(* Logix 5000 project; controller AplicacionAFEbancoDePruebas vendor 1 type 14 code 149 rev 33.12; software revision 33.01 *)

TASK MainTask (continuous, watchdog 500 ms) : MainProgram

MODULES
   Local : vendor 1 type 14 code 149 (Compact 0, rev 33.12)
      Discrete_IO : Embedded (Compact 1, rev 3.1, Output RPI 20 ms)
      PLC : 1769-L32E Ethernet Port (Ethernet 192.168.2.131, rev 20.1)
         PLC_Controller : vendor 1 type 14 code 77 (CompactLogixL32EController 0, rev 20.1, $1e2c146d$ RPI 20 ms, $44551a5c$ RPI 20 ms, $f7b069ef$ RPI 20 ms)
      VSD_AFE : vendor 1 type 143 code 8336 (Ethernet 192.168.2.50, rev 6.5, Output RPI 20 ms)
           VSD_AFE:O.LogicCommand_Stop   // Comando de Parada
           VSD_AFE:O.LogicCommand_Start   // Comando de Arranque
          : vendor 1 type 143 code 1441 (RhinoBP 10, rev 1.1)
          : vendor 1 type 143 code 416 (RhinoBP 5, rev 1.8)
          : vendor 1 type 143 code 675 (RhinoBP 13, rev 1.1)
          : vendor 1 type 143 code 416 (RhinoBP 4, rev 1.8)
          : vendor 1 type 143 code 4770 (RhinoBP 12, rev 1.1)
          : vendor 1 type 143 code 2724 (RhinoBP 14, rev 1.1)
          : vendor 1 type 143 code 767 (RhinoBP 1, rev 2.7)
END_MODULES

TYPE Dinagrama :   // Estructura para el dinagrama
STRUCT
   vPotencia : REAL[500];   // captura del vector de potencia
   vCarga : REAL[500];   // captura del vector de carga
   vPosicion : REAL[500];   // captura del vector posicion
   vProximetro : DINT[500];   // captura del vector del proximetro
   NumeroMuestras : INT;
   enabled : BOOL;
   captura : BOOL;   // Flag que indica la captura del sistema
   resetVector : BOOL;   // Flag para darle Reset al vector de posición y carga
   vEmptyREAL : REAL[500];
   vEmptyINT : DINT[500];
   tMuestreo : REAL;   // Tiempo de Muestreo de captura
END_STRUCT
END_TYPE

TYPE LSW :   // Drive - Logic Status Word
STRUCT
   Faulted : BOOL;
   Warning : BOOL;
   RunForward : BOOL;
   RunReverse : BOOL;
   Ready : BOOL;
   RemoteRef : BOOL;
   RemoteCrtl : BOOL;
   AtSpeed : BOOL;
END_STRUCT
END_TYPE

TYPE SWC :
STRUCT
   Dinagrama : Dinagrama;
   VSD : VSD;
   entradasDigitales : INT;   // Entradas Digitales
   salidasDigitales : INT;   // Salidas Digitales
   entradasAnalogas : REAL[4];   // Entradas Analogas del PLC
   salidasAnalogas : REAL[4];
END_STRUCT
END_TYPE

TYPE VSD :   // VSD
STRUCT
   VSD_O : AB:PowerFlex755T_E_31635488:O:0;
   VSD_I : AB:PowerFlex755T_E_2B0A69C5:I:0;
END_STRUCT
END_TYPE

VAR_GLOBAL   (* controller tags *)
   SRP_Displacement_Actual : REAL := 47.925312;   // Variable de Simulacion PLC DC de Desplazamiento
   SRP_Load_Actual : REAL := 10.571887;   // Variable de simulacion PLC DC de Carga
   SRP_SimActualStroke : DINT;   // Variable Simulación de PLC Variador DC
   SWC : SWC := (Dinagrama.vCarga[0] := 9.6614, Dinagrama.vCarga[1] := 9.7812, Dinagrama.vCarga[2] := 9.711983, Dinagrama.vCarga[3] := 9.725293, Dinagrama.vCarga[4] := 9.842433, Dinagrama.vCarga[5] := 9.749254, Dinagrama.vCarga[6] := 9.69601, Dinagrama.vCarga[7] := 9.7306185, Dinagrama.vCarga[8] := 9.586858, Dinagrama.vCarga[9] := 9.751916, Dinagrama.vCarga[10] := 10.223133, Dinagrama.vCarga[11] := 10.473384, Dinagrama.vCarga[12] := 10.545264, Dinagrama.vCarga[13] := 10.752919, Dinagrama.vCarga[14] := 10.928628, Dinagrama.vCarga[15] := 11.220809, Dinagrama.vCarga[16] := 11.419147, Dinagrama.vCarga[17] := 11.515653, Dinagrama.vCarga[18] := 11.572558, Dinagrama.vCarga[19] := 11.751262, Dinagrama.vCarga[20] := 11.839782, Dinagrama.vCarga[21] := 11.974224, Dinagrama.vCarga[22] := 11.854091, Dinagrama.vCarga[23] := 11.607167, Dinagrama.vCarga[24] := 11.27239, Dinagrama.vCarga[25] := 11.069394, Dinagrama.vCarga[26] := 10.880708, Dinagrama.vCarga[27] := 10.662403, Dinagrama.vCarga[28] := 10.492021, Dinagrama.vCarga[29] := 10.321636, Dinagrama.vCarga[30] := 10.193849, Dinagrama.vCarga[31] := 10.018141, Dinagrama.vCarga[32] := 9.842432, Dinagrama.vCarga[33] := 9.682698, Dinagrama.vCarga[34] := 9.586857, Dinagrama.vCarga[35] := 9.706658, Dinagrama.vCarga[36] := 9.938273, Dinagrama.vCarga[37] := 10.082034, Dinagrama.vCarga[38] := 10.241769, Dinagrama.vCarga[39] := 10.321636, Dinagrama.vCarga[40] := 10.409491, Dinagrama.vCarga[41] := 10.409491, Dinagrama.vCarga[42] := 10.457411, Dinagrama.vCarga[43] := 10.534616, Dinagrama.vCarga[44] := 10.481371, Dinagrama.vCarga[45] := 10.555914, Dinagrama.vCarga[46] := 10.705, Dinagrama.vCarga[47] := 10.603834, Dinagrama.vCarga[48] := 10.316312, Dinagrama.vCarga[49] := 10.060737, Dinagrama.vCarga[50] := 9.9223, Dinagrama.vCarga[51] := 9.850419, Dinagrama.vCarga[52] := 9.608155, Dinagrama.vCarga[53] := 9.405825, Dinagrama.vCarga[54] := 9.389851, Dinagrama.vCarga[55] := 9.230116, Dinagrama.vCarga[56] := 9.131613, Dinagrama.vCarga[57] := 9.049084, Dinagrama.vCarga[58] := 9.08103, Dinagrama.vCarga[59] := 8.9266205,
        Dinagrama.vCarga[60] := 8.873376, Dinagrama.vCarga[61] := 9.155573, Dinagrama.vCarga[62] := 9.427122, Dinagrama.vCarga[63] := 9.549585, Dinagrama.vCarga[64] := 9.682697, Dinagrama.vCarga[65] := 9.906326, Dinagrama.vCarga[66] := 10.012816, Dinagrama.vCarga[67] := 9.980869, Dinagrama.vCarga[68] := 9.996842, Dinagrama.vCarga[69] := 9.980869, Dinagrama.vCarga[70] := 10.018141, Dinagrama.vCarga[71] := 10.042101, Dinagrama.vCarga[72] := 10.098008, Dinagrama.vCarga[73] := 10.193849, Dinagrama.vCarga[74] := 9.938273, Dinagrama.vCarga[75] := 9.618804, Dinagrama.vCarga[76] := 9.546924, Dinagrama.vCarga[77] := 9.55491, Dinagrama.vCarga[78] := 9.331282, Dinagrama.vCarga[79] := 9.171547, Dinagrama.vCarga[80] := 9.347255, Dinagrama.vCarga[81] := 9.315308, Dinagrama.vCarga[82] := 9.123626, Dinagrama.vCarga[83] := 9.18752, Dinagrama.vCarga[84] := 9.331282, Dinagrama.vCarga[85] := 9.182196, Dinagrama.vCarga[86] := 9.2168045, Dinagrama.vCarga[87] := 9.565559, Dinagrama.vCarga[88] := 9.762566, Dinagrama.vCarga[89] := 9.714645, Dinagrama.vCarga[90] := 9.703996, Dinagrama.vCarga[91] := 9.842432, Dinagrama.vCarga[92] := 9.834445, Dinagrama.vCarga[93] := 9.634777, Dinagrama.vCarga[94] := 9.634777, Dinagrama.vCarga[95] := 9.656075, Dinagrama.vCarga[96] := 9.496341, Dinagrama.vCarga[97] := 9.272713, Dinagrama.vCarga[98] := 9.128951, Dinagrama.vCarga[99] := 8.910647, Dinagrama.vCarga[100] := 8.434105, Dinagrama.vCarga[101] := 8.02412, Dinagrama.vCarga[102] := 7.904319, Dinagrama.vCarga[103] := 7.78718, Dinagrama.vCarga[104] := 7.5129685, Dinagrama.vCarga[105] := 7.302651, Dinagrama.vCarga[106] := 7.281353, Dinagrama.vCarga[107] := 7.238757, Dinagrama.vCarga[108] := 6.8181233, Dinagrama.vCarga[109] := 6.6264415, Dinagrama.vCarga[110] := 6.6796865, Dinagrama.vCarga[111] := 6.903315, Dinagrama.vCarga[112] := 7.1056457, Dinagrama.vCarga[113] := 7.3771944, Dinagrama.vCarga[114] := 7.773869, Dinagrama.vCarga[115] := 7.909643, Dinagrama.vCarga[116] := 7.909643, Dinagrama.vCarga[117] := 8.077365, Dinagrama.vCarga[118] := 8.300993, Dinagrama.vCarga[119] := 8.340926,
        Dinagrama.vCarga[120] := 8.460728, Dinagrama.vCarga[121] := 8.70033, Dinagrama.vCarga[122] := 8.79617, Dinagrama.vCarga[123] := 8.788184, Dinagrama.vCarga[124] := 8.77221, Dinagrama.vCarga[125] := 8.588515, Dinagrama.vCarga[126] := 8.38086, Dinagrama.vCarga[127] := 8.340927, Dinagrama.vCarga[128] := 8.468715, Dinagrama.vCarga[129] := 8.399496, Dinagrama.vCarga[130] := 8.476701, Dinagrama.vCarga[131] := 8.532608, Dinagrama.vCarga[132] := 8.497999, Dinagrama.vCarga[133] := 8.503324, Dinagrama.vCarga[134] := 8.591178, Dinagrama.vCarga[135] := 8.56988, Dinagrama.vCarga[136] := 8.631111, Dinagrama.vCarga[137] := 8.84409, Dinagrama.vCarga[138] := 9.081031, Dinagrama.vCarga[139] := 9.278037, Dinagrama.vCarga[140] := 9.325957, Dinagrama.vCarga[141] := 9.363229, Dinagrama.vCarga[142] := 9.618804, Dinagrama.vCarga[143] := 9.682698, Dinagrama.vCarga[144] := 9.682698, Dinagrama.vCarga[145] := 9.938273, Dinagrama.vCarga[146] := 9.938273, Dinagrama.vCarga[147] := 9.938273, Dinagrama.vCarga[148] := 9.938273, Dinagrama.vCarga[149] := 9.938273, Dinagrama.vCarga[150] := 9.938273, Dinagrama.vCarga[151] := 9.938273, Dinagrama.vCarga[152] := 9.938273, Dinagrama.vCarga[153] := 9.938273, Dinagrama.vCarga[154] := 9.938273, Dinagrama.vCarga[155] := 9.938273, Dinagrama.vCarga[156] := 9.938273, Dinagrama.vCarga[157] := 9.938273, Dinagrama.vCarga[158] := 9.938273, Dinagrama.vCarga[159] := 9.938273, Dinagrama.vCarga[160] := 9.938273, Dinagrama.vCarga[161] := 9.938273, Dinagrama.vCarga[162] := 9.938273, Dinagrama.vCarga[163] := 9.938273, Dinagrama.vCarga[164] := 9.938273, Dinagrama.vCarga[165] := 9.938273, Dinagrama.vCarga[166] := 9.938273, Dinagrama.vCarga[167] := 9.938273, Dinagrama.vCarga[168] := 9.938273, Dinagrama.vCarga[169] := 9.938273, Dinagrama.vCarga[170] := 9.938273, Dinagrama.vCarga[171] := 9.938273, Dinagrama.vCarga[172] := 9.938273, Dinagrama.vCarga[173] := 9.938273, Dinagrama.vCarga[174] := 9.938273, Dinagrama.vCarga[175] := 9.938273, Dinagrama.vCarga[176] := 9.938273, Dinagrama.vCarga[177] := 9.938273, Dinagrama.vCarga[178] := 9.938273, Dinagrama.vCarga[179] := 9.938273,
        Dinagrama.vCarga[180] := 9.938273, Dinagrama.vCarga[181] := 9.938273, Dinagrama.vCarga[182] := 9.938273, Dinagrama.vCarga[183] := 9.938273, Dinagrama.vCarga[184] := 9.938273, Dinagrama.vCarga[185] := 9.938273, Dinagrama.vCarga[186] := 9.938273, Dinagrama.vCarga[187] := 9.938273, Dinagrama.vCarga[188] := 9.938273, Dinagrama.vCarga[189] := 9.938273, Dinagrama.vCarga[190] := 9.938273, Dinagrama.vCarga[191] := 9.938273, Dinagrama.vCarga[192] := 9.938273, Dinagrama.vCarga[193] := 9.938273, Dinagrama.vCarga[194] := 9.938273, Dinagrama.vCarga[195] := 9.938273, Dinagrama.vCarga[196] := 9.938273, Dinagrama.vCarga[197] := 9.938273, Dinagrama.vCarga[198] := 9.938273, Dinagrama.vCarga[199] := 9.938273, Dinagrama.vCarga[200] := 9.938273, Dinagrama.vCarga[201] := 9.938273, Dinagrama.vCarga[202] := 9.938273, Dinagrama.vCarga[203] := 9.938273, Dinagrama.vCarga[204] := 9.938273, Dinagrama.vCarga[205] := 9.938273, Dinagrama.vCarga[206] := 9.938273, Dinagrama.vCarga[207] := 9.938273, Dinagrama.vCarga[208] := 9.938273, Dinagrama.vCarga[209] := 9.938273, Dinagrama.vCarga[210] := 9.938273, Dinagrama.vCarga[211] := 9.938273, Dinagrama.vCarga[212] := 9.938273, Dinagrama.vCarga[213] := 9.938273, Dinagrama.vCarga[214] := 9.938273, Dinagrama.vCarga[215] := 9.938273, Dinagrama.vCarga[216] := 9.938273, Dinagrama.vCarga[217] := 9.938273, Dinagrama.vCarga[218] := 9.938273, Dinagrama.vCarga[219] := 9.938273, Dinagrama.vCarga[220] := 9.938273, Dinagrama.vCarga[221] := 9.938273, Dinagrama.vCarga[222] := 9.938273, Dinagrama.vCarga[223] := 9.938273, Dinagrama.vCarga[224] := 9.938273, Dinagrama.vCarga[225] := 9.938273, Dinagrama.vCarga[226] := 9.938273, Dinagrama.vCarga[227] := 9.938273, Dinagrama.vCarga[228] := 9.938273, Dinagrama.vCarga[229] := 9.938273, Dinagrama.vCarga[230] := 9.938273, Dinagrama.vCarga[231] := 10.060737, Dinagrama.vCarga[232] := 9.9223, Dinagrama.vCarga[233] := 9.7306185, Dinagrama.vCarga[234] := 9.480367, Dinagrama.vCarga[235] := 9.405825, Dinagrama.vCarga[236] := 9.389851, Dinagrama.vCarga[237] := 9.230116, Dinagrama.vCarga[238] := 9.059732, Dinagrama.vCarga[239] := 9.10499,
        Dinagrama.vCarga[240] := 9.017137, Dinagrama.vCarga[241] := 8.822793, Dinagrama.vCarga[242] := 9.0011635, Dinagrama.vCarga[243] := 9.323295, Dinagrama.vCarga[244] := 9.499002, Dinagrama.vCarga[245] := 9.549585, Dinagrama.vCarga[246] := 9.682697, Dinagrama.vCarga[247] := 10.002167, Dinagrama.vCarga[248] := 10.012816, Dinagrama.vCarga[249] := 9.980869, Dinagrama.vCarga[250] := 9.986194, Dinagrama.vCarga[251] := 9.980869, Dinagrama.vCarga[252] := 10.018141, Dinagrama.vCarga[253] := 10.042101, Dinagrama.vCarga[254] := 10.145928, Dinagrama.vCarga[255] := 10.066061, Dinagrama.vCarga[256] := 9.778539, Dinagrama.vCarga[257] := 9.578871, Dinagrama.vCarga[258] := 9.546924, Dinagrama.vCarga[259] := 9.443096, Dinagrama.vCarga[260] := 9.331282, Dinagrama.vCarga[261] := 9.259401, Dinagrama.vCarga[262] := 9.331282, Dinagrama.vCarga[263] := 9.219467, Dinagrama.vCarga[264] := 9.123626, Dinagrama.vCarga[265] := 9.18752, Dinagrama.vCarga[266] := 9.331282, Dinagrama.vCarga[267] := 9.182196, Dinagrama.vCarga[268] := 9.2168045, Dinagrama.vCarga[269] := 9.565559, Dinagrama.vCarga[270] := 9.762566, Dinagrama.vCarga[271] := 9.688023, Dinagrama.vCarga[272] := 9.746592, Dinagrama.vCarga[273] := 9.901002, Dinagrama.vCarga[274] := 9.834445, Dinagrama.vCarga[275] := 9.634777, Dinagrama.vCarga[276] := 9.634777, Dinagrama.vCarga[277] := 9.624128, Dinagrama.vCarga[278] := 9.37654, Dinagrama.vCarga[279] := 9.184858, Dinagrama.vCarga[280] := 9.046422, Dinagrama.vCarga[281] := 8.910647, Dinagrama.vCarga[282] := 8.434105, Dinagrama.vCarga[283] := 8.02412, Dinagrama.vCarga[284] := 7.851074, Dinagrama.vCarga[285] := 7.6647167, Dinagrama.vCarga[286] := 7.5129685, Dinagrama.vCarga[287] := 7.302651, Dinagrama.vCarga[288] := 7.2973266, Dinagrama.vCarga[289] := 7.1429167, Dinagrama.vCarga[290] := 6.8181233, Dinagrama.vCarga[291] := 6.6264415, Dinagrama.vCarga[292] := 6.799487, Dinagrama.vCarga[293] := 6.999156, Dinagrama.vCarga[294] := 7.2174597, Dinagrama.vCarga[295] := 7.622121, Dinagrama.vCarga[296] := 7.925617, Dinagrama.vCarga[297] := 7.909643, Dinagrama.vCarga[298] := 7.909643, Dinagrama.vCarga[299] := 8.245086,
        Dinagrama.vCarga[300] := 8.3569, Dinagrama.vCarga[301] := 8.324953, Dinagrama.vCarga[302] := 8.596502, Dinagrama.vCarga[303] := 8.70033, Dinagrama.vCarga[304] := 8.79617, Dinagrama.vCarga[305] := 8.788184, Dinagrama.vCarga[306] := 8.756237, Dinagrama.vCarga[307] := 8.588515, Dinagrama.vCarga[308] := 8.38086, Dinagrama.vCarga[309] := 8.412807, Dinagrama.vCarga[310] := 8.420794, Dinagrama.vCarga[311] := 8.431443, Dinagrama.vCarga[312] := 8.548582, Dinagrama.vCarga[313] := 8.532608, Dinagrama.vCarga[314] := 8.490012, Dinagrama.vCarga[315] := 8.559231, Dinagrama.vCarga[316] := 8.575204, Dinagrama.vCarga[317] := 8.585853, Dinagrama.vCarga[318] := 8.734939, Dinagrama.vCarga[319] := 8.84409, Dinagrama.vCarga[320] := 9.081031, Dinagrama.vCarga[321] := 9.278037, Dinagrama.vCarga[322] := 9.309984, Dinagrama.vCarga[323] := 9.554911, Dinagrama.vCarga[324] := 9.618804, Dinagrama.vCarga[325] := 9.682698, Dinagrama.vPosicion[0] := 0.22007, Dinagrama.vPosicion[1] := 0.4084145, Dinagrama.vPosicion[2] := 0.8989175, Dinagrama.vPosicion[3] := 1.5143573, Dinagrama.vPosicion[4] := 2.2604218, Dinagrama.vPosicion[5] := 3.1391559, Dinagrama.vPosicion[6] := 4.147569, Dinagrama.vPosicion[7] := 5.2654533, Dinagrama.vPosicion[8] := 6.4805126, Dinagrama.vPosicion[9] := 7.78114, Dinagrama.vPosicion[10] := 9.158964, Dinagrama.vPosicion[11] := 10.613574, Dinagrama.vPosicion[12] := 11.377348, Dinagrama.vPosicion[13] := 12.962581, Dinagrama.vPosicion[14] := 14.611691, Dinagrama.vPosicion[15] := 17.481466, Dinagrama.vPosicion[16] := 19.2797, Dinagrama.vPosicion[17] := 21.118301, Dinagrama.vPosicion[18] := 22.049511, Dinagrama.vPosicion[19] := 23.956749, Dinagrama.vPosicion[20] := 25.906015, Dinagrama.vPosicion[21] := 27.897532, Dinagrama.vPosicion[22] := 29.92443, Dinagrama.vPosicion[23] := 32.000904, Dinagrama.vPosicion[24] := 34.121273, Dinagrama.vPosicion[25] := 36.271236, Dinagrama.vPosicion[26] := 38.454124, Dinagrama.vPosicion[27] := 40.67515, Dinagrama.vPosicion[28] := 42.926197, Dinagrama.vPosicion[29] := 45.59054, Dinagrama.vPosicion[30] := 47.925312, Dinagrama.vPosicion[31] := 50.300934, Dinagrama.vPosicion[32] := 52.57733, Dinagrama.vPosicion[33] := 54.853752,
        Dinagrama.vPosicion[34] := 57.161697, Dinagrama.vPosicion[35] := 58.29858, Dinagrama.vPosicion[36] := 60.54371, Dinagrama.vPosicion[37] := 62.754997, Dinagrama.vPosicion[38] := 66.06483, Dinagrama.vPosicion[39] := 67.1463, Dinagrama.vPosicion[40] := 69.277466, Dinagrama.vPosicion[41] := 71.36186, Dinagrama.vPosicion[42] := 73.41511, Dinagrama.vPosicion[43] := 75.75438, Dinagrama.vPosicion[44] := 77.68309, Dinagrama.vPosicion[45] := 79.54948, Dinagrama.vPosicion[46] := 81.36385, Dinagrama.vPosicion[47] := 83.1282, Dinagrama.vPosicion[48] := 84.8323, Dinagrama.vPosicion[49] := 86.45127, Dinagrama.vPosicion[50] := 87.98693, Dinagrama.vPosicion[51] := 88.73018, Dinagrama.vPosicion[52] := 90.154045, Dinagrama.vPosicion[53] := 91.48115, Dinagrama.vPosicion[54] := 93.29226, Dinagrama.vPosicion[55] := 94.39419, Dinagrama.vPosicion[56] := 94.9114, Dinagrama.vPosicion[57] := 96.00089, Dinagrama.vPosicion[58] := 96.84068, Dinagrama.vPosicion[59] := 97.581314, Dinagrama.vPosicion[60] := 98.21293, Dinagrama.vPosicion[61] := 98.7474, Dinagrama.vPosicion[62] := 99.18755, Dinagrama.vPosicion[63] := 99.53332, Dinagrama.vPosicion[64] := 99.77987, Dinagrama.vPosicion[65] := 99.935196, Dinagrama.vPosicion[66] := 99.99795, Dinagrama.vPosicion[67] := 99.96849, Dinagrama.vPosicion[68] := 99.93045, Dinagrama.vPosicion[69] := 99.64918, Dinagrama.vPosicion[70] := 99.35959, Dinagrama.vPosicion[71] := 98.93282, Dinagrama.vPosicion[72] := 98.72924, Dinagrama.vPosicion[73] := 98.26827, Dinagrama.vPosicion[74] := 97.74029, Dinagrama.vPosicion[75] := 97.14606, Dinagrama.vPosicion[76] := 96.147736, Dinagrama.vPosicion[77] := 95.795845, Dinagrama.vPosicion[78] := 95.004196, Dinagrama.vPosicion[79] := 94.16693, Dinagrama.vPosicion[80] := 93.305756, Dinagrama.vPosicion[81] := 92.36308, Dinagrama.vPosicion[82] := 91.377556, Dinagrama.vPosicion[83] := 90.37801, Dinagrama.vPosicion[84] := 89.32036, Dinagrama.vPosicion[85] := 88.01027, Dinagrama.vPosicion[86] := 86.84538, Dinagrama.vPosicion[87] := 85.63856, Dinagrama.vPosicion[88] := 84.37339, Dinagrama.vPosicion[89] := 83.723206, Dinagrama.vPosicion[90] := 82.400505, Dinagrama.vPosicion[91] := 81.02402, Dinagrama.vPosicion[92] := 78.86634, Dinagrama.vPosicion[93] := 77.38295,
        Dinagrama.vPosicion[94] := 76.61854, Dinagrama.vPosicion[95] := 75.04756, Dinagrama.vPosicion[96] := 73.44262, Dinagrama.vPosicion[97] := 71.8104, Dinagrama.vPosicion[98] := 70.117615, Dinagrama.vPosicion[99] := 68.385605, Dinagrama.vPosicion[100] := 66.349724, Dinagrama.vPosicion[101] := 64.541084, Dinagrama.vPosicion[102] := 62.67875, Dinagrama.vPosicion[103] := 60.810116, Dinagrama.vPosicion[104] := 58.907894, Dinagrama.vPosicion[105] := 56.94176, Dinagrama.vPosicion[106] := 55.949615, Dinagrama.vPosicion[107] := 53.960396, Dinagrama.vPosicion[108] := 50.92777, Dinagrama.vPosicion[109] := 48.843502, Dinagrama.vPosicion[110] := 47.795254, Dinagrama.vPosicion[111] := 45.690845, Dinagrama.vPosicion[112] := 43.56501, Dinagrama.vPosicion[113] := 41.413986, Dinagrama.vPosicion[114] := 38.891975, Dinagrama.vPosicion[115] := 35.634483, Dinagrama.vPosicion[116] := 34.528854, Dinagrama.vPosicion[117] := 32.329132, Dinagrama.vPosicion[118] := 30.155361, Dinagrama.vPosicion[119] := 27.987307, Dinagrama.vPosicion[120] := 25.821117, Dinagrama.vPosicion[121] := 24.743301, Dinagrama.vPosicion[122] := 21.607874, Dinagrama.vPosicion[123] := 19.584843, Dinagrama.vPosicion[124] := 17.632542, Dinagrama.vPosicion[125] := 15.761359, Dinagrama.vPosicion[126] := 13.965392, Dinagrama.vPosicion[127] := 13.085015, Dinagrama.vPosicion[128] := 11.154951, Dinagrama.vPosicion[129] := 9.596523, Dinagrama.vPosicion[130] := 8.136012, Dinagrama.vPosicion[131] := 6.7788615, Dinagrama.vPosicion[132] := 5.529149, Dinagrama.vPosicion[133] := 4.3940463, Dinagrama.vPosicion[134] := 3.3902075, Dinagrama.vPosicion[135] := 2.520764, Dinagrama.vPosicion[136] := 1.7710685, Dinagrama.vPosicion[137] := 1.148738, Dinagrama.vPosicion[138] := 0.66532767, Dinagrama.vPosicion[139] := 0.31461334, Dinagrama.vPosicion[140] := 0.096083336, Dinagrama.vPosicion[141] := 0.009929333, Dinagrama.vPosicion[142] := 0.049646668, Dinagrama.vPosicion[143] := 0.059576, Dinagrama.vPosicion[144] := 0.059576, Dinagrama.vPosicion[145] := 60.54371, Dinagrama.vPosicion[146] := 60.54371, Dinagrama.vPosicion[147] := 60.54371, Dinagrama.vPosicion[148] := 60.54371, Dinagrama.vPosicion[149] := 60.54371, Dinagrama.vPosicion[150] := 60.54371, Dinagrama.vPosicion[151] := 60.54371, Dinagrama.vPosicion[152] := 60.54371, Dinagrama.vPosicion[153] := 60.54371,
        Dinagrama.vPosicion[154] := 60.54371, Dinagrama.vPosicion[155] := 60.54371, Dinagrama.vPosicion[156] := 60.54371, Dinagrama.vPosicion[157] := 60.54371, Dinagrama.vPosicion[158] := 60.54371, Dinagrama.vPosicion[159] := 60.54371, Dinagrama.vPosicion[160] := 60.54371, Dinagrama.vPosicion[161] := 60.54371, Dinagrama.vPosicion[162] := 60.54371, Dinagrama.vPosicion[163] := 60.54371, Dinagrama.vPosicion[164] := 60.54371, Dinagrama.vPosicion[165] := 60.54371, Dinagrama.vPosicion[166] := 60.54371, Dinagrama.vPosicion[167] := 60.54371, Dinagrama.vPosicion[168] := 60.54371, Dinagrama.vPosicion[169] := 60.54371, Dinagrama.vPosicion[170] := 60.54371, Dinagrama.vPosicion[171] := 60.54371, Dinagrama.vPosicion[172] := 60.54371, Dinagrama.vPosicion[173] := 60.54371, Dinagrama.vPosicion[174] := 60.54371, Dinagrama.vPosicion[175] := 60.54371, Dinagrama.vPosicion[176] := 60.54371, Dinagrama.vPosicion[177] := 60.54371, Dinagrama.vPosicion[178] := 60.54371, Dinagrama.vPosicion[179] := 60.54371, Dinagrama.vPosicion[180] := 60.54371, Dinagrama.vPosicion[181] := 60.54371, Dinagrama.vPosicion[182] := 60.54371, Dinagrama.vPosicion[183] := 60.54371, Dinagrama.vPosicion[184] := 60.54371, Dinagrama.vPosicion[185] := 60.54371, Dinagrama.vPosicion[186] := 60.54371, Dinagrama.vPosicion[187] := 60.54371, Dinagrama.vPosicion[188] := 60.54371, Dinagrama.vPosicion[189] := 60.54371, Dinagrama.vPosicion[190] := 60.54371, Dinagrama.vPosicion[191] := 60.54371, Dinagrama.vPosicion[192] := 60.54371, Dinagrama.vPosicion[193] := 60.54371, Dinagrama.vPosicion[194] := 60.54371, Dinagrama.vPosicion[195] := 60.54371, Dinagrama.vPosicion[196] := 60.54371, Dinagrama.vPosicion[197] := 60.54371, Dinagrama.vPosicion[198] := 60.54371, Dinagrama.vPosicion[199] := 60.54371, Dinagrama.vPosicion[200] := 60.54371, Dinagrama.vPosicion[201] := 60.54371, Dinagrama.vPosicion[202] := 60.54371, Dinagrama.vPosicion[203] := 60.54371, Dinagrama.vPosicion[204] := 60.54371, Dinagrama.vPosicion[205] := 60.54371, Dinagrama.vPosicion[206] := 60.54371, Dinagrama.vPosicion[207] := 60.54371, Dinagrama.vPosicion[208] := 60.54371, Dinagrama.vPosicion[209] := 60.54371, Dinagrama.vPosicion[210] := 60.54371, Dinagrama.vPosicion[211] := 60.54371, Dinagrama.vPosicion[212] := 60.54371, Dinagrama.vPosicion[213] := 60.54371,
        Dinagrama.vPosicion[214] := 60.54371, Dinagrama.vPosicion[215] := 60.54371, Dinagrama.vPosicion[216] := 60.54371, Dinagrama.vPosicion[217] := 60.54371, Dinagrama.vPosicion[218] := 60.54371, Dinagrama.vPosicion[219] := 60.54371, Dinagrama.vPosicion[220] := 60.54371, Dinagrama.vPosicion[221] := 60.54371, Dinagrama.vPosicion[222] := 60.54371, Dinagrama.vPosicion[223] := 60.54371, Dinagrama.vPosicion[224] := 60.54371, Dinagrama.vPosicion[225] := 60.54371, Dinagrama.vPosicion[226] := 60.54371, Dinagrama.vPosicion[227] := 60.54371, Dinagrama.vPosicion[228] := 60.54371, Dinagrama.vPosicion[229] := 60.54371, Dinagrama.vPosicion[230] := 60.54371, Dinagrama.vPosicion[231] := 86.45127, Dinagrama.vPosicion[232] := 87.98693, Dinagrama.vPosicion[233] := 89.45013, Dinagrama.vPosicion[234] := 90.82591, Dinagrama.vPosicion[235] := 92.103096, Dinagrama.vPosicion[236] := 93.29226, Dinagrama.vPosicion[237] := 94.39419, Dinagrama.vPosicion[238] := 95.391045, Dinagrama.vPosicion[239] := 96.43602, Dinagrama.vPosicion[240] := 97.23012, Dinagrama.vPosicion[241] := 97.91339, Dinagrama.vPosicion[242] := 98.4962, Dinagrama.vPosicion[243] := 98.98255, Dinagrama.vPosicion[244] := 99.37747, Dinagrama.vPosicion[245] := 99.53332, Dinagrama.vPosicion[246] := 99.77987, Dinagrama.vPosicion[247] := 99.935196, Dinagrama.vPosicion[248] := 99.99795, Dinagrama.vPosicion[249] := 99.96849, Dinagrama.vPosicion[250] := 99.8579, Dinagrama.vPosicion[251] := 99.64918, Dinagrama.vPosicion[252] := 99.35959, Dinagrama.vPosicion[253] := 98.93282, Dinagrama.vPosicion[254] := 98.49876, Dinagrama.vPosicion[255] := 98.00428, Dinagrama.vPosicion[256] := 97.44318, Dinagrama.vPosicion[257] := 96.822845, Dinagrama.vPosicion[258] := 96.147736, Dinagrama.vPosicion[259] := 95.40002, Dinagrama.vPosicion[260] := 95.004196, Dinagrama.vPosicion[261] := 94.16693, Dinagrama.vPosicion[262] := 92.83442, Dinagrama.vPosicion[263] := 91.870316, Dinagrama.vPosicion[264] := 91.377556, Dinagrama.vPosicion[265] := 90.37801, Dinagrama.vPosicion[266] := 89.32036, Dinagrama.vPosicion[267] := 88.01027, Dinagrama.vPosicion[268] := 86.84538, Dinagrama.vPosicion[269] := 85.63856, Dinagrama.vPosicion[270] := 84.37339, Dinagrama.vPosicion[271] := 83.06744, Dinagrama.vPosicion[272] := 81.722916, Dinagrama.vPosicion[273] := 80.31708,
        Dinagrama.vPosicion[274] := 78.86634, Dinagrama.vPosicion[275] := 77.38295, Dinagrama.vPosicion[276] := 76.61854, Dinagrama.vPosicion[277] := 74.24831, Dinagrama.vPosicion[278] := 72.63172, Dinagrama.vPosicion[279] := 70.97654, Dinagrama.vPosicion[280] := 69.25514, Dinagrama.vPosicion[281] := 68.385605, Dinagrama.vPosicion[282] := 66.349724, Dinagrama.vPosicion[283] := 64.541084, Dinagrama.vPosicion[284] := 61.744232, Dinagrama.vPosicion[285] := 59.862404, Dinagrama.vPosicion[286] := 58.907894, Dinagrama.vPosicion[287] := 56.94176, Dinagrama.vPosicion[288] := 54.955784, Dinagrama.vPosicion[289] := 52.964237, Dinagrama.vPosicion[290] := 50.92777, Dinagrama.vPosicion[291] := 48.843502, Dinagrama.vPosicion[292] := 46.7459, Dinagrama.vPosicion[293] := 44.632946, Dinagrama.vPosicion[294] := 42.49205, Dinagrama.vPosicion[295] := 39.97316, Dinagrama.vPosicion[296] := 37.810795, Dinagrama.vPosicion[297] := 35.634483, Dinagrama.vPosicion[298] := 34.528854, Dinagrama.vPosicion[299] := 31.23504, Dinagrama.vPosicion[300] := 29.075682, Dinagrama.vPosicion[301] := 26.898933, Dinagrama.vPosicion[302] := 24.743301, Dinagrama.vPosicion[303] := 23.68875, Dinagrama.vPosicion[304] := 21.607874, Dinagrama.vPosicion[305] := 19.584843, Dinagrama.vPosicion[306] := 16.676949, Dinagrama.vPosicion[307] := 15.761359, Dinagrama.vPosicion[308] := 13.965392, Dinagrama.vPosicion[309] := 12.251199, Dinagrama.vPosicion[310] := 10.367658, Dinagrama.vPosicion[311] := 8.857708, Dinagrama.vPosicion[312] := 7.4485517, Dinagrama.vPosicion[313] := 6.144711, Dinagrama.vPosicion[314] := 4.950763, Dinagrama.vPosicion[315] := 3.8806663, Dinagrama.vPosicion[316] := 2.945591, Dinagrama.vPosicion[317] := 2.1355166, Dinagrama.vPosicion[318] := 1.448219, Dinagrama.vPosicion[319] := 1.148738, Dinagrama.vPosicion[320] := 0.66532767, Dinagrama.vPosicion[321] := 0.31461334, Dinagrama.vPosicion[322] := 0.038433332, Dinagrama.vPosicion[323] := 0.03971733, Dinagrama.vPosicion[324] := 0.049646668, Dinagrama.vPosicion[325] := 0.059576, Dinagrama.vProximetro[0] := 1, Dinagrama.vProximetro[1] := 1, Dinagrama.vProximetro[2] := 1, Dinagrama.NumeroMuestras := 143, Dinagrama.tMuestreo := 0.05, VSD.VSD_O.P10_VRefAStpt := 37.3, VSD.VSD_I.DriveStatus := 2#0010_0001_0000_0000_0000_0100_0000_1101, VSD.VSD_I.DriveStatus_Ready := 1,
        VSD.VSD_I.DriveStatus_CommandDir := 1, VSD.VSD_I.DriveStatus_ActualDir := 1, VSD.VSD_I.DriveStatus_SpdRefBit0 := 1, VSD.VSD_I.DriveStatus_AtZeroSpeed := 1, VSD.VSD_I.DriveStatus_EnableOn := 1, VSD.VSD_I.P10_VRefCommanded := 59.407898, VSD.VSD_I.DCBusVolts := 707.12067, VSD.VSD_I.P10_HeatsnkTemp := 20.0, VSD.VSD_I.ElapsedRunTime := 29.436, VSD.VSD_I.LastFaultCode := 13002, VSD.VSD_I.ElapsedkWH := -20501, entradasDigitales := 3, entradasAnalogas[0] := -1.7e-44, entradasAnalogas[1] := -9.176336e+29, entradasAnalogas[2] := 3.8693e-41, entradasAnalogas[3] := 6.66079e-40, salidasAnalogas[0] := 1.e-45, salidasAnalogas[1] := 6.e-45, salidasAnalogas[2] := 4.e-45);
        .Dinagrama.enabled   // Habilitar Adquision
END_VAR

PROGRAM MainProgram   (* main routine R000_MainRoutine *)
VAR
   Captura : BOOL;
   contadorAux : ALIAS FOR counter[0].ACC;
   counter : COUNTER[10];
   Enabled : BOOL;
   Flag : BOOL;
   habilitar : DINT;
   myoneshot : BOOL[32];
        [0]   // oneshot toogle bot dinagrama
        [1]   // oneshor reset del ocntador
        [2]   // reset de la flag cuando se habilita y se deshabilita
   Proximetro_Virtual : ALIAS FOR SRP_SimActualStroke;
   SPM_Reference : REAL := 8.5;
   timer : TIMER[10] := ([0].PRE := 50);
        [0]   // Tiempo Muestreo
END_VAR

ROUTINE R000_MainRoutine   (* ladder *)
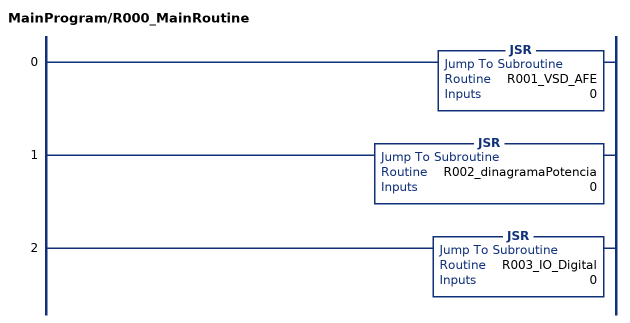
   0: JSR(R001_VSD_AFE,0);
   1: JSR(R002_dinagramaPotencia,0);
   2: JSR(R003_IO_Digital,0);
END_ROUTINE

ROUTINE R001_VSD_AFE   (* ladder *)
// Comandos Basicos de Operación de VSD AFE
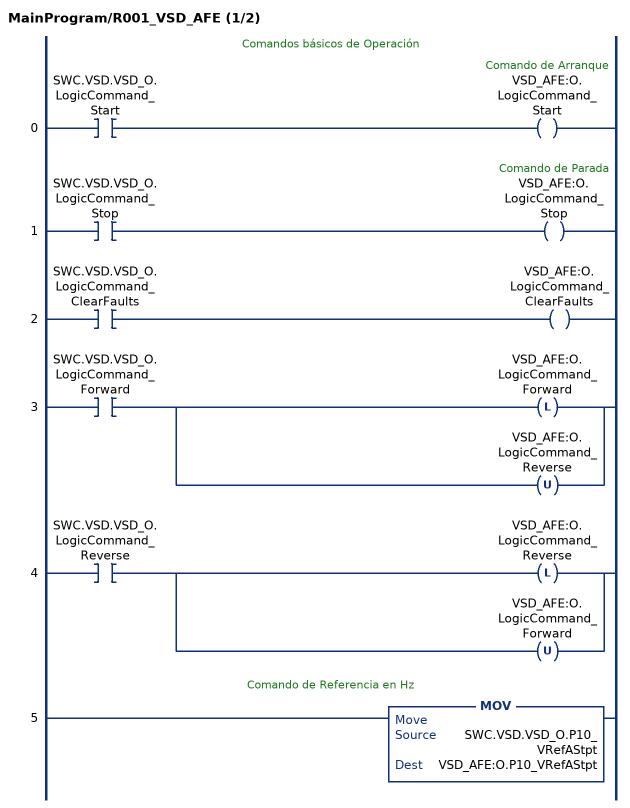
   // Comandos básicos de Operación
   0: XIC(SWC.VSD.VSD_O.LogicCommand_Start)OTE(VSD_AFE:O.LogicCommand_Start);
   1: XIC(SWC.VSD.VSD_O.LogicCommand_Stop)OTE(VSD_AFE:O.LogicCommand_Stop);
   2: XIC(SWC.VSD.VSD_O.LogicCommand_ClearFaults)OTE(VSD_AFE:O.LogicCommand_ClearFaults);
   3: XIC(SWC.VSD.VSD_O.LogicCommand_Forward)[OTL(VSD_AFE:O.LogicCommand_Forward) ,OTU(VSD_AFE:O.LogicCommand_Reverse) ];
   4: XIC(SWC.VSD.VSD_O.LogicCommand_Reverse)[OTL(VSD_AFE:O.LogicCommand_Reverse) ,OTU(VSD_AFE:O.LogicCommand_Forward) ];
   // Comando de Referencia en Hz
   5: MOV(SWC.VSD.VSD_O.P10_VRefAStpt,VSD_AFE:O.P10_VRefAStpt);
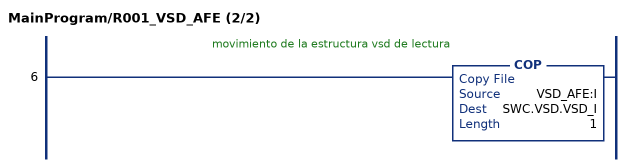
   // movimiento de la estructura vsd de lectura
   6: COP(VSD_AFE:I,SWC.VSD.VSD_I,1);
END_ROUTINE

ROUTINE R002_dinagramaPotencia   (* ladder *)
// Adquisión de los diferentes strokes para la captura del dinagrama de superficie
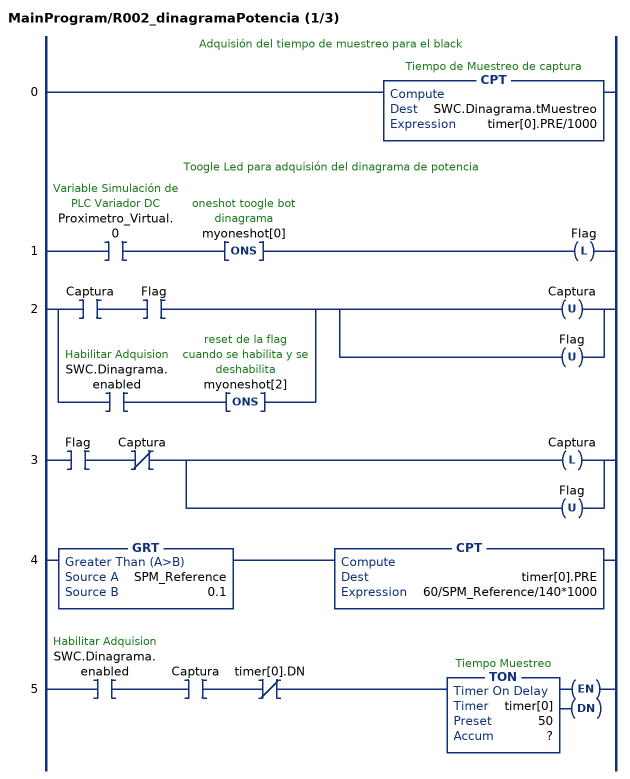
   // Adquisión del tiempo de muestreo para el black
   0: CPT(SWC.Dinagrama.tMuestreo,timer[0].PRE/1000);
   // Toogle Led para adquisión del dinagrama de potencia
   1: XIC(Proximetro_Virtual.0)ONS(myoneshot[0])OTL(Flag);
   2: [XIC(Captura) XIC(Flag) ,XIC(SWC.Dinagrama.enabled) ONS(myoneshot[2]) ][OTU(Captura) ,OTU(Flag) ];
   3: XIC(Flag)XIO(Captura)[OTL(Captura) ,OTU(Flag) ];
   4: GRT(SPM_Reference,0.1)CPT(timer[0].PRE,60/SPM_Reference/140*1000);
   5: XIC(SWC.Dinagrama.enabled)XIC(Captura)XIO(timer[0].DN)TON(timer[0],?,?);
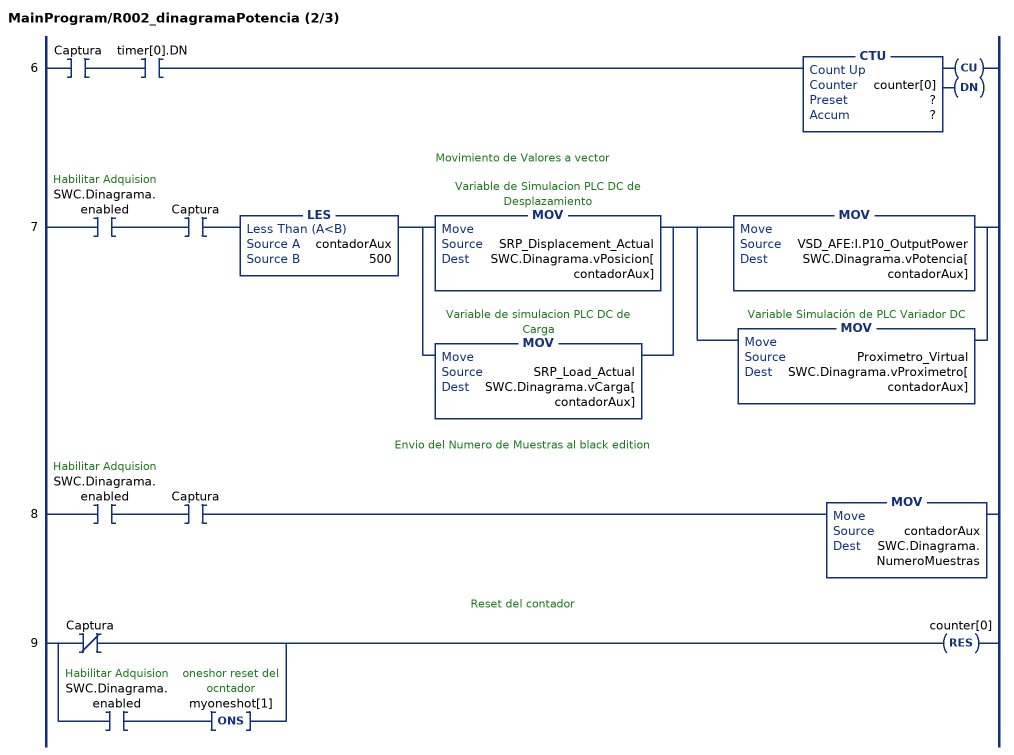
   6: XIC(Captura)XIC(timer[0].DN)CTU(counter[0],?,?);
   // Movimiento de Valores a vector
   7: XIC(SWC.Dinagrama.enabled)XIC(Captura)LES(contadorAux,500)[MOV(SRP_Displacement_Actual,SWC.Dinagrama.vPosicion[contadorAux]) ,MOV(SRP_Load_Actual,SWC.Dinagrama.vCarga[contadorAux]) ][MOV(VSD_AFE:I.P10_OutputPower,SWC.Dinagrama.vPotencia[contadorAux]) ,MOV(Proximetro_Virtual,SWC.Dinagrama.vProximetro[contadorAux]) ];
   // Envio del Numero de Muestras al black edition
   8: XIC(SWC.Dinagrama.enabled)XIC(Captura)MOV(contadorAux,SWC.Dinagrama.NumeroMuestras);
   // Reset del contador
   9: [XIO(Captura) ,XIC(SWC.Dinagrama.enabled) ONS(myoneshot[1]) ]RES(counter[0]);
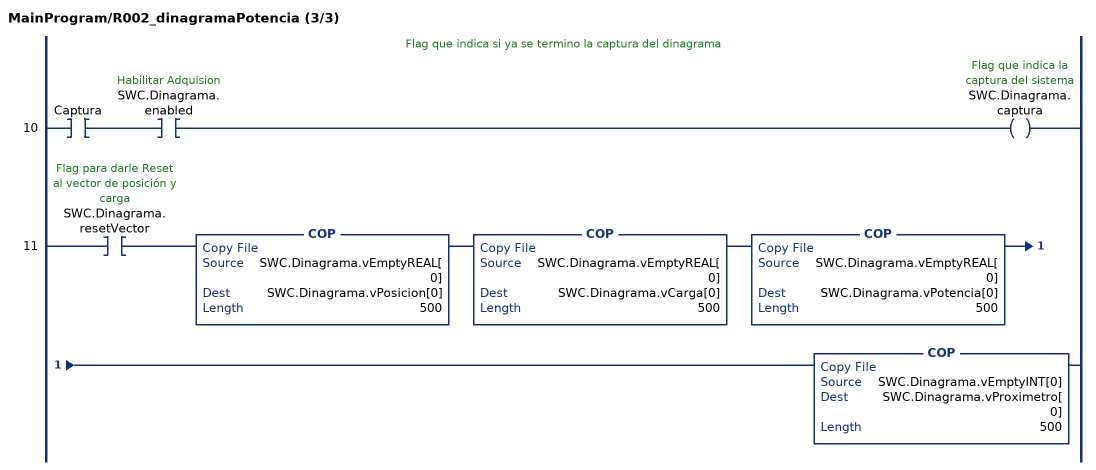
   // Flag que indica si ya se termino la captura del dinagrama
   10: XIC(Captura)XIC(SWC.Dinagrama.enabled)OTE(SWC.Dinagrama.captura);
   11: XIC(SWC.Dinagrama.resetVector)COP(SWC.Dinagrama.vEmptyREAL[0],SWC.Dinagrama.vPosicion[0],500)COP(SWC.Dinagrama.vEmptyREAL[0],SWC.Dinagrama.vCarga[0],500)COP(SWC.Dinagrama.vEmptyREAL[0],SWC.Dinagrama.vPotencia[0],500)COP(SWC.Dinagrama.vEmptyINT[0],SWC.Dinagrama.vProximetro[0],500);
END_ROUTINE

ROUTINE R003_IO_Digital   (* ladder *)
// Entradas Digitales
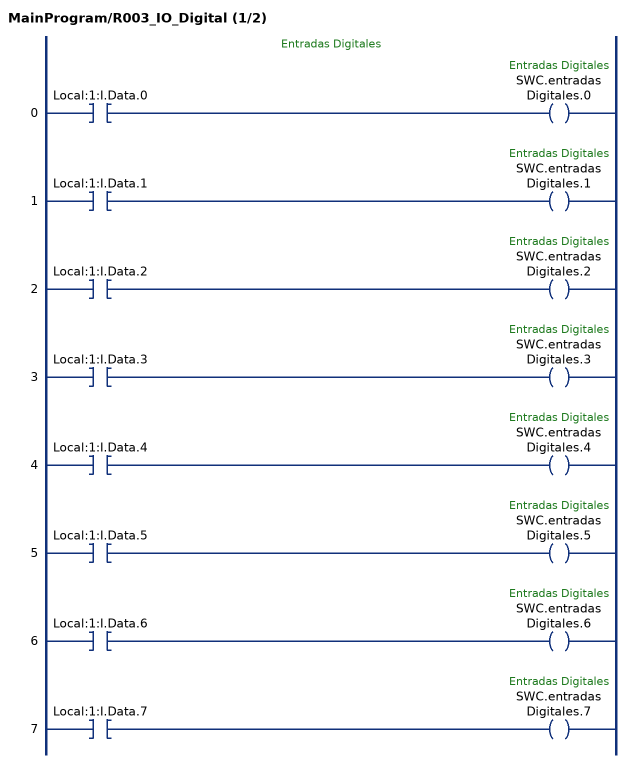
   // Entradas Digitales
   0: XIC(Local:1:I.Data.0)OTE(SWC.entradasDigitales.0);
   1: XIC(Local:1:I.Data.1)OTE(SWC.entradasDigitales.1);
   2: XIC(Local:1:I.Data.2)OTE(SWC.entradasDigitales.2);
   3: XIC(Local:1:I.Data.3)OTE(SWC.entradasDigitales.3);
   4: XIC(Local:1:I.Data.4)OTE(SWC.entradasDigitales.4);
   5: XIC(Local:1:I.Data.5)OTE(SWC.entradasDigitales.5);
   6: XIC(Local:1:I.Data.6)OTE(SWC.entradasDigitales.6);
   7: XIC(Local:1:I.Data.7)OTE(SWC.entradasDigitales.7);
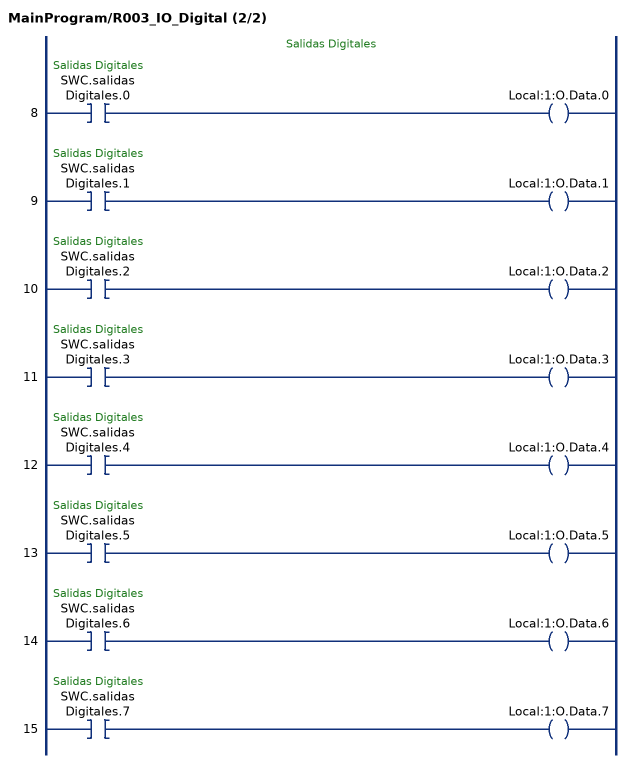
   // Salidas Digitales
   8: XIC(SWC.salidasDigitales.0)OTE(Local:1:O.Data.0);
   9: XIC(SWC.salidasDigitales.1)OTE(Local:1:O.Data.1);
   10: XIC(SWC.salidasDigitales.2)OTE(Local:1:O.Data.2);
   11: XIC(SWC.salidasDigitales.3)OTE(Local:1:O.Data.3);
   12: XIC(SWC.salidasDigitales.4)OTE(Local:1:O.Data.4);
   13: XIC(SWC.salidasDigitales.5)OTE(Local:1:O.Data.5);
   14: XIC(SWC.salidasDigitales.6)OTE(Local:1:O.Data.6);
   15: XIC(SWC.salidasDigitales.7)OTE(Local:1:O.Data.7);
END_ROUTINE
END_PROGRAM
